TYPE WcStateInputToggleBase_F68C23A9 :
STRUCT
END_STRUCT
END_TYPE

(* stored: Version 1.2.0.0, ProductVersion 3.1.4024.9
   DUT WcStateInputToggleBase_F68C23A9: Id {b265616c-c7ec-4bb3-bfcc-18705089cbbc} *)
